FUNCTION_BLOCK "Driver_Working"   // FB15, SCL
{ S7_Optimized_Access := 'TRUE' }
VERSION : 0.1
   VAR_INPUT
      in_bStartButtonPushed : Bool;
      in_bEnableReturnTask : Bool;   // Включение. Режима добора задания
      in_bCountTriesReset : Bool;   // Сброс количества попыток перекладки
      in_usiCountTries : USInt;   // Количество попыток выполнить задание
      in_iRequired : Int;   // Задание. Кол-во материала
      in_bAlarm : Bool;   // Наличие Аварии
      in_bAlarmReset : Bool;   // Сброс Аварии
      in_bInHome : Bool;   // Сигнал от робота. Робот в Домашней позиции
      in_bProgReq : Bool;   // Сигнал от робота. Запрос на новую программу
      in_bResume : Bool;   // Продолжить выполнения задания
      in_bCancelTask : Bool;   // Отмена задания
      in_bModeDebug : Bool;   // Режим. Отладки
      in_pointer_array : Array[0..1] of Bool;
   END_VAR
   VAR_OUTPUT
      out_bStart : Bool;   // Команда Старт
      out_bStop : Bool;   // Команда Стоп
      out_usiProgrammNumber : USInt;   // Номер программы
      out_uiZoneFrom : UInt;   // Задание. Откуда забирать материал
      out_uiZoneTo : UInt;   // Задание. Куда класть материал
      out_uiRequired : UInt;   // Задание. Кол-во материала
      out_A_bCantWork : Bool;   // Авария Робот не может продолжать работу
      out_usiCountTries : USInt;   // Количество попыток
      out_strJobStatus : String[15];   // Статус задачи
   END_VAR
   VAR_IN_OUT
      in_Task : "TypeRobotTask";   // Собранное задание
      in_usiTaskStatus : UInt;   // Состояние Задания
      in_bDebugNextStep : Bool;   // Режим отладки. Следующий шаг
   END_VAR
   VAR
      _bStart : Bool;   // Бит старта Робота
      _bStop : Bool;   // Бит стоп Робота
      _uiZoneFrom : UInt;   // Задание. Откуда забирать материал
      _uiZoneTo : UInt;   // Задание. Куда класть материал
      _uiRequired : Int;   // Задание. Кол-во материала
      _bCancelTask : Bool;
      _usiStatus : USInt;
      _uiProgrammNumber : UInt;   // Номер программы
      _usiLastProgrammNumber : USInt;   // Последний номер программы
      _usiCountTries : USInt;   // Счетчик попыток
      _usiCountTriesHeight : USInt;
      _usiStepRegularWork : USInt;
      tStepBHX_scan : Array[0..17] of TON_TIME;
      i_tStepBHX_scan : USInt;
      tStepRegularWork : Array[0..17] of TON_TIME;
      i_tStepRegularWork : USInt;
      _usiStepCancelTask : USInt;
      tStepCancelTask : Array[0..17] of TON_TIME;
      i_tStepCancelTask : USInt;
      _usiStepAlaram : USInt;
      tStepAlaram : Array[0..17] of TON_TIME;
      i_tStepAlaram : USInt;
      rtFinish : R_TRIG;   // Тригер окончания задания
      rtAlarmReset : R_TRIG;   // Тригер продолжения задания
      rtCountTries : R_TRIG;   // Тригер счетчик попыток выполнения задания
      rtCountTriesReset : R_TRIG;   // Тригер сброса попыток выполнения задания
      rtStartButtonPushed : R_TRIG;
      _robot_status_ok : Bool;
      _part_status_ok : Bool;
      _task_status_ok : Bool;
      _robot_signals_ok : Bool;
      _first_step_ok : Bool;
      _act_done : Bool;
      _select_done : Bool;
      _task_id_ok : Bool;
      _lrobot_task_id : LInt;
   END_VAR
   VAR CONSTANT
      cTaskStatus_Ready : USInt := 0;   // Статус задания. Готов
      cTaskStatus_NewTaskReceived : USInt := 1;   // Статус задания. Получено новое задание
      cTaskStatus_InProcess : USInt := 2;   // Статус задания. В процессе
      cTaskStatus_Finished : USInt := 3;   // Статус задания. Закончено
      cWorkStatus_RegularWork : USInt := 99;   // Режим. Нормальная работа
      cWorkStatus_CancelTask : USInt := 1;   // Режим. Возврат в дом
      cWorkStatus_Alarm : USInt := 0;   // Режим. Авария
      cStep_ReadyForNewCyrcle : USInt := 0;   // Готовностьи к новому циклу
      cStep_SetRegularWorkProgramm : USInt := 1;   // Изменяем номер программы
      cStep_StartBitUp : USInt := 2;   // Выставляем стартовый бит
      cStep_StartBitDown : USInt := 3;   // Снимаем стартовый бит
      cStep_InProcess : USInt := 4;   // Переводим состояние задания в вПроцессе
      cStep_TaskFinish : USInt := 5;   // Задание завершенно
      cStep_DelayBeforeHome : USInt := 6;   // Ждем новое задание перед отправкой в дом
      cStep_SetGoHomeProgramm : USInt := 7;   // Отправляем робота в дом
      cStep_StartBitUpGoHome : USInt := 8;   // Выставляем стартовый бит
      cStep_StartBitDownGoHome : USInt := 9;   // Снимаем стартовый бит
      cStep_SendStopUp : USInt := 11;   // Выставляем Стоповый бит
      cStep_SendStopDown : USInt := 12;   // Снимаем Стоповый бит
      cStep_SetInitProgramm : USInt := 13;
      cStep_SetDeInitProgramm : USInt := 14;
      cStep_SetPostCorrProgramm : USInt := 15;
      cStep_StopBitUpGoHome : USInt := 16;
      cStep_StopBitDownGoHome : USInt := 17;
      cWorkStatus_Scanning : USInt := 2;   // Режим. Сканирование поддона
      cWorkStatus_HeightMeasuring : USInt := 3;
      cWorkStatus_Gripping_in : USInt := 4;
      cWorkStatus_Loading : USInt := 5;
      cWorkStatus_Unoading : USInt := 6;
      cWorkStatus_Flipping : USInt := 7;
      cWorkStatus_Dropping_out : USInt := 8;
      cWorkStatus_BHX_load : USInt := 9;
      cWorkStatus_BHX_unload : USInt := 10;
      cWorkStatus_BHX_scan : USInt := 11;
      cWorkStatus_test_BHX_load : USInt := 12;
      cWorkStatus_test_BHX_unload : USInt := 13;
      cWorkStatus_POS_load : USInt := 14;
      cWorkStatus_POS_unload : USInt := 15;
      cWorkStatus_Gripping_buf : USInt := 16;
      cWorkStatus_Dropping_buf : USInt := 17;
      cWorkStatus_Gripping_flip : USInt := 18;
      cWorkStatus_Dropping_flip : USInt := 19;
      cRange_k : Real := 0.0405;
      cRange_b : Real := 213.0;
   END_VAR
BEGIN
   ////////////////////////////Защиты и Блокировки////////////////////////////
   //Счетчик попыток на выполнение задания
   #rtCountTries(CLK := #_usiStepRegularWork = 1);
   IF #rtCountTries.Q THEN
       #_usiCountTries := #_usiCountTries + 1;
       #_usiCountTriesHeight := #_usiCountTriesHeight + 1;
   END_IF;
   #rtCountTriesReset(CLK := #in_bCountTriesReset);
   #rtAlarmReset(CLK := #in_bResume);
   IF #rtCountTriesReset.Q OR #rtAlarmReset.Q THEN
       #_usiCountTries := 0;
       #_usiCountTriesHeight := 0;
       #out_A_bCantWork := FALSE;
   END_IF;
   IF #_usiCountTries > (#in_usiCountTries) THEN
       #out_A_bCantWork := TRUE;
   END_IF;
   ///////////////////////////////////////////////////////////////////////////


   //
   #rtStartButtonPushed(CLK := #in_bStartButtonPushed AND (#_usiStepRegularWork < 1 OR #_usiStepRegularWork > 4));
   IF #rtStartButtonPushed.Q THEN
       #in_usiTaskStatus := 1;
   END_IF;

   //////////////////////////////Выбор состояния//////////////////////////////
   IF #in_bAlarm THEN
       //Статус: Авария 
       #_usiStatus := #cWorkStatus_Alarm;
   ELSIF (#in_bCancelTask OR #_bCancelTask) AND NOT #in_bAlarm THEN
       //Статус: Возврат в Дом 
       #_usiStatus := #cWorkStatus_CancelTask;
   ELSIF #in_bProgReq AND NOT #_bCancelTask AND NOT #in_bAlarm THEN //AND "PLC_AutoFeedingModeActive" THEN
       //Статус. Нормальный режим работы
       #_usiStatus := #cWorkStatus_RegularWork;
   ELSE
       #_uiProgrammNumber := 0;
   END_IF;
   ///////////////////////////////////////////////////////////////////////////

   ///////////////////////////////Логика работы///////////////////////////////
   //Статус: Нормальный режим работы
   IF #_usiStatus = #cWorkStatus_RegularWork THEN
       #rtFinish(CLK := #in_bProgReq);

       #_first_step_ok:=(#tStepRegularWork[#cStep_DelayBeforeHome].ET > T#20ms
                           OR #_usiStepRegularWork = #cStep_ReadyForNewCyrcle
                           OR (#_usiStepRegularWork = #cStep_SetRegularWorkProgramm AND #_uiProgrammNumber=0)
                           OR #tStepRegularWork[#cStep_StartBitDownGoHome].ET >= T#5s
                           OR "Robot"."EXT_FIRST_START")
                           AND #in_bProgReq
                           AND NOT "Robot"."PRO_MOVE_KRC";
                           #_task_status_ok := "RobotTasks".Robot1.task_status = 'received' OR "RobotTasks".Robot1.task_status = 'on_trajectory'
                           ;//OR "RobotTasks".Robot1.task_status = 'new_trajectory';
                           #_robot_status_ok := ("RobotTasks".Robot1.robot_status <> 'unknown') AND "RobotTasks".Robot1.robot_status <> 'manual_mode' AND "RobotTasks".Robot1.robot_status <> 'busy';
                           #_part_status_ok := ("RobotTasks".Robot1.part_status <> 'scanned'  OR "RobotTasks".Robot1.operation_type='measuring_height') AND "RobotTasks".Robot1.part_status <> 'done';

                           #_robot_signals_ok := "Robot"."USER_SAF_KRC" AND "Robot"."ALARM_STOP_KRC"  AND "Robot"."PERI_RDY_KRC" AND NOT "Robot"."STOPMESS_KRC" AND NOT "To_KUKA_PLC_STOP";

       #_task_id_ok:=#_lrobot_task_id="RobotTasks".Robot1.robot_task_id;

       //Шаг: Готовность
       IF #_first_step_ok AND #_task_status_ok AND #_robot_status_ok AND #_part_status_ok
           AND NOT #_select_done THEN
           #_lrobot_task_id := "RobotTasks".Robot1.robot_task_id;
           #_usiStepRegularWork := #cStep_ReadyForNewCyrcle;
       END_IF;

       //Шаг: Изменяем номер программы
       IF  // #rtFinish.Q AND
           #tStepRegularWork[#cStep_ReadyForNewCyrcle].ET > T#20ms AND
           #in_bProgReq THEN
           #_usiStepRegularWork := #cStep_SetRegularWorkProgramm;
       END_IF;

       //Шаг: Выставляем стартовый бит
       IF #tStepRegularWork[#cStep_SetRegularWorkProgramm].ET > T#20ms 
           AND #_uiProgrammNumber>0
           //machine shunt
           AND (NOT "RobotTasks".Robot1."w/o_machine_mode"
           OR ("RobotTasks".Robot1.robot_trajectory <> 'LoadMachine' OR "RobotTasks".Robot1.robot_trajectory <> 'UnloadMachine' )
           //OR (#_uiProgrammNumber<>7 AND #_uiProgrammNumber<>8)
           )
           //#_usiStepRegularWork = #cStep_SetRegularWorkProgramm AND
           AND #in_bProgReq THEN
           #_usiStepRegularWork := #cStep_StartBitUp;
       END_IF;

       //Шаг: Снимаем стартовый бит
       IF #tStepRegularWork[#cStep_StartBitUp].ET > T#20ms
           THEN

               #_usiStepRegularWork := #cStep_StartBitDownGoHome;
       END_IF;

       //Шаг: Переводим состояние задания в вПроцессе
       IF #tStepRegularWork[#cStep_StartBitDownGoHome].ET > T#20ms 
           AND NOT #in_bProgReq
           //AND "RobotTasks".Robot1.robot_status <> 'home'
       THEN
           #_usiStepRegularWork := #cStep_InProcess;
           #_act_done := FALSE;
       END_IF;

       //Шаг: Переводим состояние задания в в начало
       IF (#tStepRegularWork[#cStep_StartBitDownGoHome].ET >= T#1m
           //machine shunt
           OR (#tStepRegularWork[#cStep_InProcess].ET >= T#1ms AND "RobotTasks".Robot1."w/o_machine_mode"))
           AND #in_bProgReq AND "RobotTasks".Robot1.robot_alarm_reset
       THEN
           #_usiStepRegularWork := #cStep_ReadyForNewCyrcle;
       END_IF;

       //Шаг: Задание завершенно
       IF (#tStepRegularWork[#cStep_InProcess].ET > T#20ms
           //machine shunt
           OR ("RobotTasks".Robot1."w/o_machine_mode" AND ("RobotTasks".Robot1.robot_trajectory = 'LoadMachine' OR "RobotTasks".Robot1.robot_trajectory = 'UnloadMachine')
           //OR ("RobotTasks".Robot1."w/o_machine_mode" AND (#_uiProgrammNumber=7 OR #_uiProgrammNumber=8)
                   AND #tStepRegularWork[#cStep_SetRegularWorkProgramm].ET > T#20ms
               ))
               AND #in_bProgReq
               //AND ROR(IN := "Robot"."PGNO_REFL_KRC", N := 8) = #_uiProgrammNumber
       THEN
           #_usiStepRegularWork := #cStep_TaskFinish;
           #_act_done := FALSE;
       END_IF;

       //Шаг: Переход к ожиданию нового цикла
       IF  #tStepRegularWork[#cStep_TaskFinish].ET > T#500ms OR "To_KUKA_PLC_STOP" THEN
           #_usiStepRegularWork := #cStep_DelayBeforeHome;
           #_uiProgrammNumber := 0;
       END_IF;

       CASE #_usiStepRegularWork OF
           #cStep_ReadyForNewCyrcle:
               //Шаг: Готовность
               #_bStart := FALSE;
               #_uiProgrammNumber := 0;

           #cStep_SetRegularWorkProgramm:
               //Шаг: Изменяем номер программы
               IF #_uiProgrammNumber = 0 THEN
                   "Get_Robot_Program"(in_Task:="RobotTasks".Robot1, Program_number=>#_uiProgrammNumber );
                   IF #_uiProgrammNumber <> 0 THEN
                       IF "RobotTasks".Robot1.part_status = 'ordered' THEN
                           "To_KUKA_Part_Destination" := 1;
                       ELSIF "RobotTasks".Robot1.part_status = 'processing' THEN
                           "To_KUKA_Part_Destination" := 2;
                       ELSIF "RobotTasks".Robot1.part_status = 'loading' THEN
                           "To_KUKA_Part_Destination" := 3;
                       ELSIF "RobotTasks".Robot1.part_status = 'unloading' THEN
                           "To_KUKA_Part_Destination" := 4;
                       ELSIF "RobotTasks".Robot1.part_status = 'done' THEN
                           "To_KUKA_Part_Destination" := 5;
                       ELSIF "RobotTasks".Robot1.part_status = 'in_machine' THEN
                           "To_KUKA_Part_Destination" := 6;
                       ELSIF "RobotTasks".Robot1.part_status = 'pallet_in' THEN
                           "To_KUKA_Part_Destination" := 7;
                       ELSIF "RobotTasks".Robot1.part_status = 'pallet_buf' THEN
                           "To_KUKA_Part_Destination" := 8;
                       ELSIF "RobotTasks".Robot1.part_status = 'pallet_out' THEN
                           "To_KUKA_Part_Destination" := 9;
                       ELSIF "RobotTasks".Robot1.part_status = 'gripper' THEN
                           "To_KUKA_Part_Destination" := 10;
                       ELSIF "RobotTasks".Robot1.part_status = 'grabbing' THEN
                           "To_KUKA_Part_Destination" := 11;
                       ELSIF "RobotTasks".Robot1.part_status = 'dropping' THEN
                           "To_KUKA_Part_Destination" := 12;
                       ELSIF "RobotTasks".Robot1.part_status = 'scanning' THEN
                           "To_KUKA_Part_Destination" := 13;
                       ELSIF "RobotTasks".Robot1.part_status = 'part_slot' THEN
                           "To_KUKA_Part_Destination" := 14;
                       ELSIF "RobotTasks".Robot1.part_status = 'flip_table' THEN
                           "To_KUKA_Part_Destination" := 15;
                       ELSIF "RobotTasks".Robot1.part_status = 'flipping' THEN
                           "To_KUKA_Part_Destination" := 16;
                       ELSIF "RobotTasks".Robot1.part_status = 'scanned' THEN
                           "To_KUKA_Part_Destination" := 17;
                       ELSIF "RobotTasks".Robot1.part_status = 'measuring' THEN
                           "To_KUKA_Part_Destination" := 18;
                       END_IF;
                       "RobotTasks".Robot1.robot_program:=#_uiProgrammNumber;
                       "RobotTasks".Robot1.robot_trajectory:="Robot_Programs".List[#_uiProgrammNumber].trajectory;
                       //"RobotTasks".Robot1.task_status:='new_trajectory';
                   END_IF;
               END_IF;

           #cStep_StartBitUp:
               //Шаг: Выставляем стартовый бит
               #_bStart := TRUE;

           #cStep_StartBitDownGoHome:
               //Шаг: Снимаем стартовый бит
               #_bStart := FALSE;

           #cStep_InProcess:
               //Шаг: Переводим состояние задания в вПроцессе
               IF "RobotTasks".Robot1.robot_trajectory = 'PartHeightMeasuring' AND
                   #tStepRegularWork[#cStep_InProcess].ET > T#200ms AND NOT "Robot"."PRO_MOVE_KRC" THEN
                   "RobotTasks".Robot1.part_pos_Z := "Robot".POS_ACT_Z - ("InGripperRangefinder" * #cRange_k + #cRange_b);
                   "RobotTasks".Robot1.slot_pos_Z := ("InGripperRangefinder" * #cRange_k + #cRange_b);
               END_IF;
               IF "Robot_Programs".List["RobotTasks".Robot1.robot_program].OUT_Status.inprocess_part_status = '' THEN
                   CASE "Robot"."Part_Status" OF
                       1:  "RobotTasks".Robot1.part_status := 'ordered';
                       2:  "RobotTasks".Robot1.part_status := 'processing';
                       3:  "RobotTasks".Robot1.part_status := 'loading';
                       4:  "RobotTasks".Robot1.part_status := 'unloading';
                       5:  "RobotTasks".Robot1.part_status := 'done';
                       6:  "RobotTasks".Robot1.part_status := 'in_machine';
                       7:  "RobotTasks".Robot1.part_status := 'pallet_in';
                       8:  "RobotTasks".Robot1.part_status := 'pallet_buf';
                       9:  "RobotTasks".Robot1.part_status := 'pallet_out';
                       10: "RobotTasks".Robot1.part_status := 'gripper';
                       11: "RobotTasks".Robot1.part_status := 'grabbing';
                       12: "RobotTasks".Robot1.part_status := 'dropping';
                       13: "RobotTasks".Robot1.part_status := 'scanning';
                       14: "RobotTasks".Robot1.part_status := 'part_slot';
                       15: "RobotTasks".Robot1.part_status := 'flip_table';
                       16: "RobotTasks".Robot1.part_status := 'flipping';
                       17: "RobotTasks".Robot1.part_status := 'scanned';
                       18: "RobotTasks".Robot1.part_status := 'measuring';
                   END_CASE;
               END_IF;

               IF NOT #_act_done AND #_robot_signals_ok AND #_task_id_ok THEN
                   //IF "RobotTasks".Robot1.robot_trajectory = 'PutOnSlot' THEN
                   //"RobotTasks".Robot1.part_slot := "RobotTasks".Robot1.free_slot;
                   //END_IF;
                   "RobotTasks".Robot1.task_status := "Robot_Programs".List["RobotTasks".Robot1.robot_program].OUT_Status.inprocess_task_status;
                   IF "Robot_Programs".List["RobotTasks".Robot1.robot_program].OUT_Status.inprocess_part_status <> '' THEN
                       "RobotTasks".Robot1.part_status := "Robot_Programs".List["RobotTasks".Robot1.robot_program].OUT_Status.inprocess_part_status;
                   END_IF;
                   #_act_done := TRUE;
               END_IF;

           #cStep_TaskFinish:
               //Шаг: Задание завершенно
               IF NOT #_act_done AND #_robot_signals_ok AND #_task_id_ok THEN
                   IF "RobotTasks".Robot1.robot_trajectory = 'PutOnFlipTableB' OR "RobotTasks".Robot1.robot_trajectory = 'AutoMachiningA_' THEN
                       IF "RobotTasks".Robot1.part_side = 'A' THEN
                           "RobotTasks".Robot1.part_side := 'B';
                       ELSIF "RobotTasks".Robot1.part_side = 'B' THEN
                           "RobotTasks".Robot1.part_side := 'A';
                       END_IF;
                   END_IF;
                   IF "RobotTasks".Robot1.robot_trajectory = 'PartHeightMeasuring' THEN
                       "RobotTasks".Robot1.part_pos_Z := "Robot".POS_ACT_Z - ("InGripperRangefinder" * #cRange_k + #cRange_b);
                       "RobotTasks".Robot1.slot_pos_Z := ("InGripperRangefinder" * #cRange_k + #cRange_b);
                   END_IF;
                   IF "RobotTasks".Robot1.robot_trajectory = 'Pallet_Scanning' THEN
                       "Matrix_output".scan_lay_number := "Matrix_output".scan_lay_number + 1;
                   END_IF;
                   IF "RobotTasks".Robot1.robot_trajectory = 'TakeFromSlot' THEN
                       "RobotTasks".Robot1.part_slot := 0;
                   END_IF;
                   //Не тот слой
                   IF "RobotTasks".Robot1.robot_trajectory = 'TakeFromPalletIn' AND NOT "Robot"."PartOK" THEN
                       //"RobotTasks".Robot1.task_status := 'not_sended';
                       //"RobotTasks".Robot1.part_status := 'ordered';
                       ;
                   END_IF;
                   "RobotTasks".Robot1.task_status := "Robot_Programs".List["RobotTasks".Robot1.robot_program ].OUT_Status.finish_task_status;
                   IF "Robot_Programs".List["RobotTasks".Robot1.robot_program].OUT_Status.finish_part_status <> '' THEN
                       "RobotTasks".Robot1.part_status := "Robot_Programs".List["RobotTasks".Robot1.robot_program].OUT_Status.finish_part_status;
                    END_IF;
                   #_act_done := TRUE;
               END_IF;
       END_CASE;
   END_IF;

   //Статус: Отмена задания и возврат в дом
   IF #_usiStatus = #cWorkStatus_CancelTask THEN
       //Шаг: Отправляем на робота команду стоп (для выхода из программы)
       IF #_usiStepCancelTask = #cStep_ReadyForNewCyrcle OR #in_bCancelTask THEN
           #_usiStepCancelTask := #cStep_SendStopUp;
       END_IF;

       //Шаг: Снимаем команду стоп
       IF #tStepCancelTask[#cStep_SendStopUp].ET > T#300ms THEN
           #_usiStepCancelTask := #cStep_SendStopDown;
       END_IF;

       //Шаг: Изменяем номер программы
       IF #tStepCancelTask[#cStep_SendStopDown].ET > T#200ms THEN
           #_usiStepCancelTask := #cStep_SetGoHomeProgramm;
       END_IF;

       //Шаг: Отправляем стартовый бит
       IF #tStepCancelTask[#cStep_SetGoHomeProgramm].ET > T#300ms THEN
           #_usiStepCancelTask := #cStep_StartBitUpGoHome;
       END_IF;

       //Шаг: Снимаем стартовый бит
       IF #tStepCancelTask[#cStep_StartBitUpGoHome].ET > T#300ms OR #in_bInHome THEN
           #_usiStepCancelTask := #cStep_StartBitDownGoHome;
       END_IF;

       CASE #_usiStepCancelTask OF
           #cStep_SendStopUp:
               //Шаг: Отправляем на робота команду стоп(для выхода из программы в CELL) и сбрасываем вакуум
               #_bStop := TRUE;
               #_bCancelTask := TRUE;

           #cStep_SendStopDown:
               //Шаг: Снимаем команду стоп и срос вакуума
               #_bStop := FALSE;

           #cStep_SetGoHomeProgramm:
               //Шаг: Изменяем номер программы
               #_uiProgrammNumber := 10;

           #cStep_StartBitUpGoHome:
               //Шаг: Отправляем стартовый бит
               #_bStart := TRUE;

           #cStep_StartBitDownGoHome:
               //Шаг: Снимаем стартовый бит
               #_bStart := FALSE;
               #_bCancelTask := FALSE;
       END_CASE;
   ELSE
       #_usiStepCancelTask := 0;
       #_bCancelTask := FALSE;
       #_bStop := FALSE;
   END_IF;

   //Статус: Авария, Возврат в дом
   IF #_usiStatus = #cWorkStatus_Alarm THEN
       //Шаг: Изменяем номер программы
       IF  #_usiStepAlaram = 0 AND #in_bAlarmReset THEN
           #_usiStepAlaram := #cStep_SetGoHomeProgramm;
       END_IF;

       //Шаг: Отправляем стартовый бит
       IF #tStepAlaram[#cStep_SetGoHomeProgramm].ET > T#20ms THEN
           #_usiStepAlaram := #cStep_StartBitUpGoHome;
       END_IF;

       //Шаг: Снимаем стартовый бит
       IF #tStepAlaram[#cStep_StartBitUpGoHome].ET > T#20msTHEN
           #_usiStepAlaram := #cStep_StartBitDownGoHome;
       END_IF;

       CASE #_usiStepAlaram OF
           #cStep_SetGoHomeProgramm:
               //Шаг: Изменяем номер программы
               #_uiProgrammNumber := 100;

           #cStep_StartBitUpGoHome:
               //Шаг: Отправляем стартовый бит
               #_bStart := TRUE;

           #cStep_StartBitDownGoHome:
               //Шаг: Снимаем стартовый бит
               #_bStart := FALSE;
       END_CASE;
   ELSE
       #_usiStepAlaram := 0;
   END_IF;

   ///////////////////////////////////////////////////////////////////////////

   ///////////////////////////////Запись выходов//////////////////////////////
   IF #_uiProgrammNumber<>0 THEN
       #_usiLastProgrammNumber := #_uiProgrammNumber;
   END_IF;
   #out_usiProgrammNumber := #_uiProgrammNumber;
   #out_bStart := #_bStart;
   #out_bStop := #_bStop;
   #out_uiZoneFrom := #_uiZoneFrom;
   #out_uiZoneTo := #_uiZoneTo;
   #out_uiRequired := #_uiRequired;
   #out_usiCountTries := #_usiCountTries;
   ///////////////////////////////////////////////////////////////////////////

   //////////////////////////////////Таймеры//////////////////////////////////
   //Запуск
   #tStepRegularWork[#_usiStepRegularWork](IN := TRUE,
                                           PT := T#1m);
   #tStepCancelTask[#_usiStepCancelTask](IN := TRUE,
                                             PT := T#1m);
   #tStepAlaram[#_usiStepAlaram](IN := TRUE,
                                 PT := T#1m);
   //Сброс
   FOR #i_tStepRegularWork := 0 TO 17 DO
       IF #_usiStepRegularWork <> #i_tStepRegularWork THEN
           #tStepRegularWork[#i_tStepRegularWork](IN := FALSE,
                                                  PT := T#10s);
       END_IF;
   END_FOR;
   FOR #i_tStepCancelTask := 0 TO 15 DO
       IF #_usiStepCancelTask <> #i_tStepCancelTask THEN
           #tStepCancelTask[#i_tStepCancelTask](IN := FALSE,
                                                PT := T#10s);
       END_IF;
   END_FOR;
   FOR #i_tStepAlaram := 0 TO 15 DO
       IF #_usiStepAlaram <> #i_tStepAlaram THEN
           #tStepAlaram[#i_tStepAlaram](IN := FALSE,
                                        PT := T#10s);
       END_IF;
   END_FOR;
   ///////////////////////////////////////////////////////////////////////////
END_FUNCTION_BLOCK

// folder: 5_Matrix_scanner

FUNCTION_BLOCK "DADProtocol"   // FB2, SCL
{ S7_Optimized_Access := 'TRUE' }
VERSION : 0.1
   VAR_INPUT
      DAD_ENABLE : Bool;
      IOconditioning_Enable : Bool;   // User should edit this parameter according to the Reader configuration in DL.CODE
      DataConsistency_Enable : Bool;   // User should edit this parameter according to the Reader configuration in DL.CODE
      OutputExArea_FirstByteAddress : Int;   // User should edit this parameter according to the Reader Output Exchange area addresses
      OutputExArea_Size : Int;   // User should edit this parameter according to the Reader Output Exchange area size
      InputExArea_FirstByteAddress : Int;   // User should edit this parameter according to the Reader Input Exchange area addresses
      InputExArea_Size : Int;   // User should edit this parameter according to the Reader Input Exchange area size
   END_VAR
   VAR_OUTPUT
      newDataBlockReceived : Bool;
      newDataBlockLength : Int;
   END_VAR
   VAR_IN_OUT
      Do_Resync : Bool;
      Do_SendData : Bool;
      DataToSendLength : Byte;
   END_VAR
   VAR
      newInputDataAvailable : Bool;
      InputExArea_Type : Byte := 16#81;   // User should edit this parameter according to the Reader Input Exchange area type. 16#81 --> Input ; 16#82 --> Output ; 16#84 --> DB
      OutputExArea_Type : Byte := 16#82;   // User should edit this parameter according to the Reader Output Exchange area type. 16#81 --> Input ; 16#82 --> Output ; 16#84 --> DB
      DB_Number : DInt;   // If the Exchange Area type is 16#84 (DB), this parameter specifies the DB number
      inputBuffer : Array[0..512] of Byte;
      outputBuffer : Array[0..512] of Byte;
      DAD_PRTL_FIRST_ITERATION : Bool := true;
      DAD_InternalStates : Int;
      AddressOffset : Int;
      InputDataLenByteAddress : Int;
      InputControlByteAddress : Int;
      InputFirstDataByteAddress : Int;
      InputDataConistencyByteAddress : Int;
      InputDataByteAddress : Int;
      InputDataAvailable_Actual : Bool;
      InputFragmentedData_Actual : Bool;
      InputFragmentedData_Previous : Bool;
      InputDeviceDadEnable : Bool;
      InputResyncAck : Bool;
      InputControlByte : Byte;
      InputDataLength : Byte;
      InputDataConsistencyByte : Byte;
      DataByteIndex : Int;
      OutputControlByteAddress : Int;
      OutputControlByte : Byte;
      OutputDataConsistencyByteAddress : Int;
      OutputAckDataReceived : Bool;
      TempByteValue : Byte;
      BufferDataByteIndex : Int;
      BeginFragmentedDataRx : Bool;
      EndFragmentedDataRx : Bool;
      FragmentedDataRxEnable : Bool;
      DataFragmentIndex : Int;
      MaxInputFragmentDimension : Int;
      DAD_PRTL_NUM_BYTE : Int;
      IO_COND_NUM_BYTE : Int;
      DATA_CONSISTENCY_NUM_BYTE : Int;
      Error_INPUT_DATA_CONSISTENCY : Bool;
      Error_DAD_DISABLED_ON_DEVICE : Bool;
      OutputDataLenByteAddress : Int;
      OutputFirstDataByteAddress : Int;
      NewMessageReady : Bool;
      ackDataReceived : Bool;
   END_VAR
   VAR_TEMP
      MessageByteIndex : Int;
      resetByte : Byte;
   END_VAR
   VAR CONSTANT
      IDLE : Int := 0;
      WAIT_DEVICE_DAD_ENABLING : Int := 1;
      CHECK_DATA_CONSISTENCY : Int := 10;
      READ_DATA : Int := 20;
      SEND_DATA : Int := 40;
      WAIT_ACK_DATA_SENT : Int := 41;
      SEND_SYNC_REQUEST : Int := 30;
      WAIT_SYNC_ACK : Int := 31;
      SEND_END_SYNC_REQUEST : Int := 32;
      WAIT_END_SYNC_ACK : Int := 33;
   END_VAR
BEGIN
   IF #DAD_ENABLE THEN
       // IF THE DAD PROTOCOL IS ENABLED..

       IF #DAD_PRTL_FIRST_ITERATION THEN

           // ONLY DURING THE FIRST ITERATION AFTER DAD PROTOCOL ENABLING...

           (*------------------------------------------------------------------------------
           ********************* PROTOCOL INITIALIZATION PHASE ****************************
           --------------------------------------------------------------------------------

           The Protocol initializes its parameters AND sets the Bit 7 of the Output Control
           Byte.

           ================================================================================
           Depending on the configuration parameters the addresses of the Protocol Bytes 
           varies. Suppose an Exchange Area of N Bytes. If DAD, I/O condtioning, and Data
           Consistency are enabled then the position of the bytes inside the data frame 
           will be the following.

               BYTEs POSITIONs     BYTEs Desriptions  

           |         0         | I/0 Conditioning      |
           |         1         | DAD CTRL Byte         |
           |         2         | DAD SAP Byte          |
           |         3         | DAD LENGTH Byte       |
           |      4 -> N-2     | DATA                  |
           |        N-1        | DATA CONSISTENCY Byte |

           ================================================================================*)

           #DAD_PRTL_NUM_BYTE              := 3;

           IF #IOconditioning_Enable THEN
               // If I/O conditioning is actiated the I/O data is shifted forward by one byte
               #IO_COND_NUM_BYTE           := 1;
           END_IF;

           IF #DataConsistency_Enable THEN
               // If I/O conditioning is actiated the last Byte of the Exchange area will
               // contain the copy of the DAD Control Byte
               #DATA_CONSISTENCY_NUM_BYTE          := 1;
               #InputDataConistencyByteAddress     := #InputExArea_FirstByteAddress + #InputExArea_Size - 1;
               #OutputDataConsistencyByteAddress   := #OutputExArea_FirstByteAddress + #OutputExArea_Size - 1;
           END_IF;

           // Effective dimension of the data which can be received
           #MaxInputFragmentDimension      := #InputExArea_Size - #IO_COND_NUM_BYTE - #DATA_CONSISTENCY_NUM_BYTE - #DAD_PRTL_NUM_BYTE;

           #InputControlByteAddress        := #InputExArea_FirstByteAddress + #IO_COND_NUM_BYTE;
           #InputDataLenByteAddress        := #InputExArea_FirstByteAddress + #IO_COND_NUM_BYTE + 2;
           #InputFirstDataByteAddress      := #InputExArea_FirstByteAddress + #IO_COND_NUM_BYTE + 3;
           #OutputControlByteAddress       := #OutputExArea_FirstByteAddress + #IO_COND_NUM_BYTE;
           #OutputDataLenByteAddress       := #OutputExArea_FirstByteAddress + #IO_COND_NUM_BYTE + 2;
           #OutputFirstDataByteAddress     := #OutputExArea_FirstByteAddress + #IO_COND_NUM_BYTE + 3;

           // DAD Output Bit Enable set to '1' by the protocol
           POKE_BOOL(area                  := #OutputExArea_Type,
                     byteOffset            := #OutputControlByteAddress,
                     bitOffset             := 7,
                     dbNumber              := #DB_Number,
                     value                 := TRUE);

           #newDataBlockReceived           := FALSE;
           #newDataBlockLength             := 0;

           #DAD_PRTL_FIRST_ITERATION       := FALSE;

           // !!! After enabling the DAD, the PLC performs a resynchronization with the device !!!
           #DAD_InternalStates             := #SEND_SYNC_REQUEST;

       ELSE

           // IF IT'S NOT THE FIRST ITERATION AFTER DAD PROTOCOL ENABLING....

           (* =================================================================================
           ------------------------------------------------------------------------------------

           1st Operation.                INPUT/OUTPUT SAMPLING 

           ----------------------------------------------------------------------------------
           ==================================================================================*)

           // Storing the Actual Values of the INPUT CONTROL BYTE's BITS OF INTEREST  

           #InputControlByte               := PEEK_BYTE(area := #InputExArea_Type, byteOffset := #InputControlByteAddress, dbNumber := #DB_Number);
           #InputDataAvailable_Actual      := #InputControlByte.%X0;
           #InputResyncAck                 := #InputControlByte.%X2;
           #InputFragmentedData_Actual     := #InputControlByte.%X3;
           #InputDeviceDadEnable           := #InputControlByte.%X7;
           #InputDataConsistencyByte       := PEEK_BYTE(area := #InputExArea_Type, byteOffset := #InputDataConistencyByteAddress, dbNumber := #DB_Number);

           // Storing the Actual Values of the OUTPUT CONTROL BYTE's BITS OF INTEREST
           #OutputControlByte              := PEEK_BYTE(area := #OutputExArea_Type, byteOffset := #OutputControlByteAddress, dbNumber := #DB_Number);
           #OutputAckDataReceived          := #OutputControlByte.%X0;
           //my huck
           //#InputResyncAck := FALSE;
           (*==================================================================================
           ++++++++++++++++++++++++++++++++++++++++++++++++++++++++++++++++++++++++++++++++++++

           2nd Operation.           BEGIN DAD FINITE STATES MACHINE

           ++++++++++++++++++++++++++++++++++++++++++++++++++++++++++++++++++++++++++++++++++++
           ==================================================================================*)

           CASE #DAD_InternalStates OF

                   (* ------------------------------------------------------------------------------------------
                   ********************************** PROTOCOL IDLE STATE **************************************
                   ---------------------------------------------------------------------------------------------

                   In the IDLE state the Protocol controls the input of the function block and the input control
                   Byte to determin which procedure has to be done *)

               0: // IDLE

                   // ========================= CHECK FOR NEW INPUT DATA =============================

                   #newInputDataAvailable              := #InputDataAvailable_Actual <> #OutputAckDataReceived;

                   IF #newInputDataAvailable THEN
                       // If a new Stream Of Data is available from the reader..
                       // Rising Edge of the Bit 3 in the Input CTRL Byte means Start Of FRAGMENTED Data Trasmission
                       #BeginFragmentedDataRx          := #InputFragmentedData_Actual AND NOT #InputFragmentedData_Previous;
                       // Falling Edge of the Bit 3 in the Input CTRL Byte means End Of FRAGMENTED Data Trasmission
                       #EndFragmentedDataRx            := NOT #InputFragmentedData_Actual AND #InputFragmentedData_Previous;

                       IF #BeginFragmentedDataRx THEN
                           // If the Data is Fragmented the Protocol prepares for receiving each fragment
                           #FragmentedDataRxEnable     := TRUE;
                           #DataFragmentIndex          := 0;
                       END_IF;

                       IF #DataConsistency_Enable THEN

                           // Protocol Verifies the consistency and THEN read the data
                           IF #InputControlByte = #InputDataConsistencyByte THEN
                               #Error_INPUT_DATA_CONSISTENCY       := FALSE;
                               #DAD_InternalStates                 := #READ_DATA;
                           ELSE
                               #Error_INPUT_DATA_CONSISTENCY       := TRUE;
                               // #DAD_InternalStates                 := #CHECK_DATA_CONSISTENCY;
                           END_IF;

                       ELSE

                           // Protocol Reads the data
                           #DAD_InternalStates                     := #READ_DATA;

                       END_IF;

                   END_IF;

                   #InputFragmentedData_Previous := #InputFragmentedData_Actual;


                   (*========================= USER ASKED FOR SENDING DATA ==========================
                      The Send Data procedure has higher priority than the reading data one
                   *)

                   IF #Do_SendData THEN
                       #DAD_InternalStates := #SEND_DATA;
                   END_IF;



                   (*=========================== USER ASKED FOR RESYNC ==============================
                      The Resynchronization procedure has higher priority than sending/reading data
                   *)

                   IF #Do_Resync THEN
                       #DAD_InternalStates                 := #SEND_SYNC_REQUEST;
                   END_IF;

                   (*=========================== DAD ON DEVICE IS OFF ===============================
                   If the device is down the protocol waits for its recover (DAD Bit sets to 1) and
                   automatically resync with it
                   *)

                   IF NOT #InputDeviceDadEnable THEN
                       #Error_DAD_DISABLED_ON_DEVICE       := TRUE;
                       #DAD_InternalStates                 := #WAIT_DEVICE_DAD_ENABLING;
                   END_IF;


                   (* --------------------------------------------------------------------------------------
                   ************************* PROTOCOL WAITS FOR DEVICE RECOVER *****************************
                   ----------------------------------------------------------------------------------------*)

               1: // WAIT_DEVICE_DAD_ENABLING

                   IF #InputDeviceDadEnable THEN
                       #Error_DAD_DISABLED_ON_DEVICE       := FALSE;
                       #DAD_InternalStates                 := #SEND_SYNC_REQUEST;
                   END_IF;


                   (* --------------------------------------------------------------------------------------
                   ******************************* PROTOCOL RECEIVES DATA ***********************************
                   ----------------------------------------------------------------------------------------*)

               20: // READ_DATA

                   #InputDataLength := PEEK_BYTE(area := #InputExArea_Type, byteOffset := #InputDataLenByteAddress, dbNumber := #DB_Number);

                   FOR #DataByteIndex := 0 TO BYTE_TO_INT(#InputDataLength) - 1 DO
                       #InputDataByteAddress           := #InputFirstDataByteAddress + #DataByteIndex;
                       #TempByteValue                  := PEEK_BYTE(area := #InputExArea_Type, byteOffset := #InputDataByteAddress, dbNumber := #DB_Number);
                       #BufferDataByteIndex            := #DataByteIndex + (#MaxInputFragmentDimension * #DataFragmentIndex);
                       #inputBuffer[#BufferDataByteIndex] := #TempByteValue;
                   END_FOR;

                   IF #FragmentedDataRxEnable THEN
                       // If the Fragmentation is Enabled i prepare for reading the next fragment
                       #DataFragmentIndex := #DataFragmentIndex + 1;

                       IF #EndFragmentedDataRx THEN
                           // If it has been received the last fragment the Protocol:
                           #newDataBlockReceived   := NOT #newDataBlockReceived;
                           #newDataBlockLength     := #BufferDataByteIndex + 1;
                           #FragmentedDataRxEnable := FALSE;       // Disable the Data Fragmentation Enable
                           #DataFragmentIndex      := 0;           // Reset the Data Fragment Index
                       END_IF;

                   ELSE
                       #newDataBlockReceived       := NOT #newDataBlockReceived;
                       #newDataBlockLength         := #BufferDataByteIndex + 1;
                   END_IF;

                   // SEND_ACKNOWLEDGE_DATA_READ

                   POKE_BOOL(area          := #OutputExArea_Type,
                             byteOffset    := #OutputControlByteAddress,
                             bitOffset     := 0,
                             dbNumber      := #DB_Number,
                             value         := #InputDataAvailable_Actual); // DAD Protocol send the Ack

                   #DAD_InternalStates     := #IDLE;

                   (* --------------------------------------------------------------------------------------
                   ************************* PROTOCOL RESYNCHRONIZES WITH DEVICE ***************************
                   ---------------------------------------------------------------------------------------*)

               30: // SEND_SYNC_REQUEST

                   POKE_BOOL(area          := #OutputExArea_Type,
                             byteOffset    := #OutputControlByteAddress,
                             bitOffset     := 2,
                             dbNumber      := #DB_Number,
                             value         := TRUE); // Protocol SET the Sync REQUEST

                   #DAD_InternalStates     := #WAIT_SYNC_ACK;

               31: // WAIT_SYNC_ACK

                   //Protocol Waits the Acknowledge from the Reader
                   IF #InputResyncAck THEN

                       POKE_BOOL(area          := #OutputExArea_Type,
                                 byteOffset    := #OutputControlByteAddress,
                                 bitOffset     := 1,
                                 dbNumber      := #DB_Number,
                                 value         := FALSE); // Protocol RESET the Output Data Ready Bit

                       POKE_BOOL(area          := #OutputExArea_Type,
                                 byteOffset    := #OutputControlByteAddress,
                                 bitOffset     := 0,
                                 dbNumber      := #DB_Number,
                                 value         := FALSE); // Protocol RESET the Input Data Received Bit

                       #DAD_InternalStates     := #SEND_END_SYNC_REQUEST;

                   END_IF;

               32: // SEND_END_SYNC_REQUEST

                   POKE_BOOL(area              := #OutputExArea_Type,
                             byteOffset        := #OutputControlByteAddress,
                             bitOffset         := 2,
                             dbNumber          := #DB_Number,
                             value             := FALSE); // Protocol RESET the Sync REQUEST

                   #DAD_InternalStates := #WAIT_END_SYNC_ACK;

               33: // WAIT_END_SYNC_ACK

                   IF NOT #InputResyncAck THEN
                       #Do_Resync       := FALSE;           // Reset the Resync command, so that operation is executed just one time
                       #DAD_InternalStates     := #IDLE;
                   END_IF;


                   (* --------------------------------------------------------------------------------------
                   ******************************** PROTOCOL SENDS DATA ************************************
                   ----------------------------------------------------------------------------------------*)

               40: // SEND_DATA

                   POKE(area := #OutputExArea_Type,
                        byteOffset := #OutputDataLenByteAddress,
                        dbNumber := 0,
                        value := #DataToSendLength);

                   FOR #MessageByteIndex := 0 TO BYTE_TO_INT(#DataToSendLength)-1 DO
                       POKE(area := #OutputExArea_Type,
                            byteOffset := #OutputFirstDataByteAddress + #MessageByteIndex,
                            dbNumber := 0,
                            value := #outputBuffer[#MessageByteIndex]);
                   END_FOR;

                   #NewMessageReady := NOT #NewMessageReady;

                   POKE_BOOL(area := #OutputExArea_Type,
                             byteOffset := #OutputControlByteAddress,
                             bitOffset := 1,
                             dbNumber := 0,
                             value := #NewMessageReady);

                   #DAD_InternalStates := 41;

               41: // WAIT_ACK_DATA_SENT

                   #ackDataReceived := PEEK_BOOL(area := #InputExArea_Type, dbNumber := 0, byteOffset := #InputControlByteAddress, bitOffset := 1);

                   IF #ackDataReceived = #NewMessageReady THEN
                       #Do_SendData := FALSE;
                       #DAD_InternalStates := #IDLE;
                   END_IF;



           END_CASE;// END STATES MACHINE

           (*==================================================================================
           ++++++++++++++++++++++++++++++++++++++++++++++++++++++++++++++++++++++++++++++++++++

                                      END DAD FINITE STATES MACHINE

           ++++++++++++++++++++++++++++++++++++++++++++++++++++++++++++++++++++++++++++++++++++
           ==================================================================================*)

       END_IF;// END FIRST ITERATION IF

       IF #DataConsistency_Enable THEN
           // IF DATA CONSISTENCY IS ENBLED:
           // The DAD Protocol copies the DAD CTRL Byte to the last byte position in the Out Exchange area.
           #OutputControlByte      := PEEK_BYTE(area := #OutputExArea_Type, byteOffset := #OutputControlByteAddress, dbNumber := #DB_Number);
           POKE(area               := #OutputExArea_Type,
                byteOffset         := #OutputDataConsistencyByteAddress,
                dbNumber           := #DB_Number,
                value              := #OutputControlByte);
       END_IF;

   ELSIF NOT #DAD_ENABLE & NOT #DAD_PRTL_FIRST_ITERATION THEN // IF THE DAD PROTOCOL IS DISABLED

       #resetByte              := 2#0000_0000;
       POKE(   area            := #OutputExArea_Type,
               byteOffset      := #OutputControlByteAddress,
               dbNumber        := #DB_Number,
               value           := #resetByte);

       #Do_Resync := FALSE;
       #Do_SendData := FALSE;
       #newDataBlockReceived := FALSE;
       #newDataBlockLength := 0;

       #DAD_PRTL_FIRST_ITERATION := TRUE;

   END_IF;// END DAD ENABLE IF
END_FUNCTION_BLOCK

FUNCTION "Matrix" : Void   // FC2, LAD
{ S7_Optimized_Access := 'TRUE' }
VERSION : 0.1
   VAR_TEMP
      RetVal : Word;
      PhaseON : DWord;
      PhaseOFF : DWord;
   END_VAR
   VAR_TEMP   // added for the SCL form of the ladder/FBD networks
      _w1 : Bool;
      _w2 : Bool;
   END_VAR
BEGIN

REGION Network 1
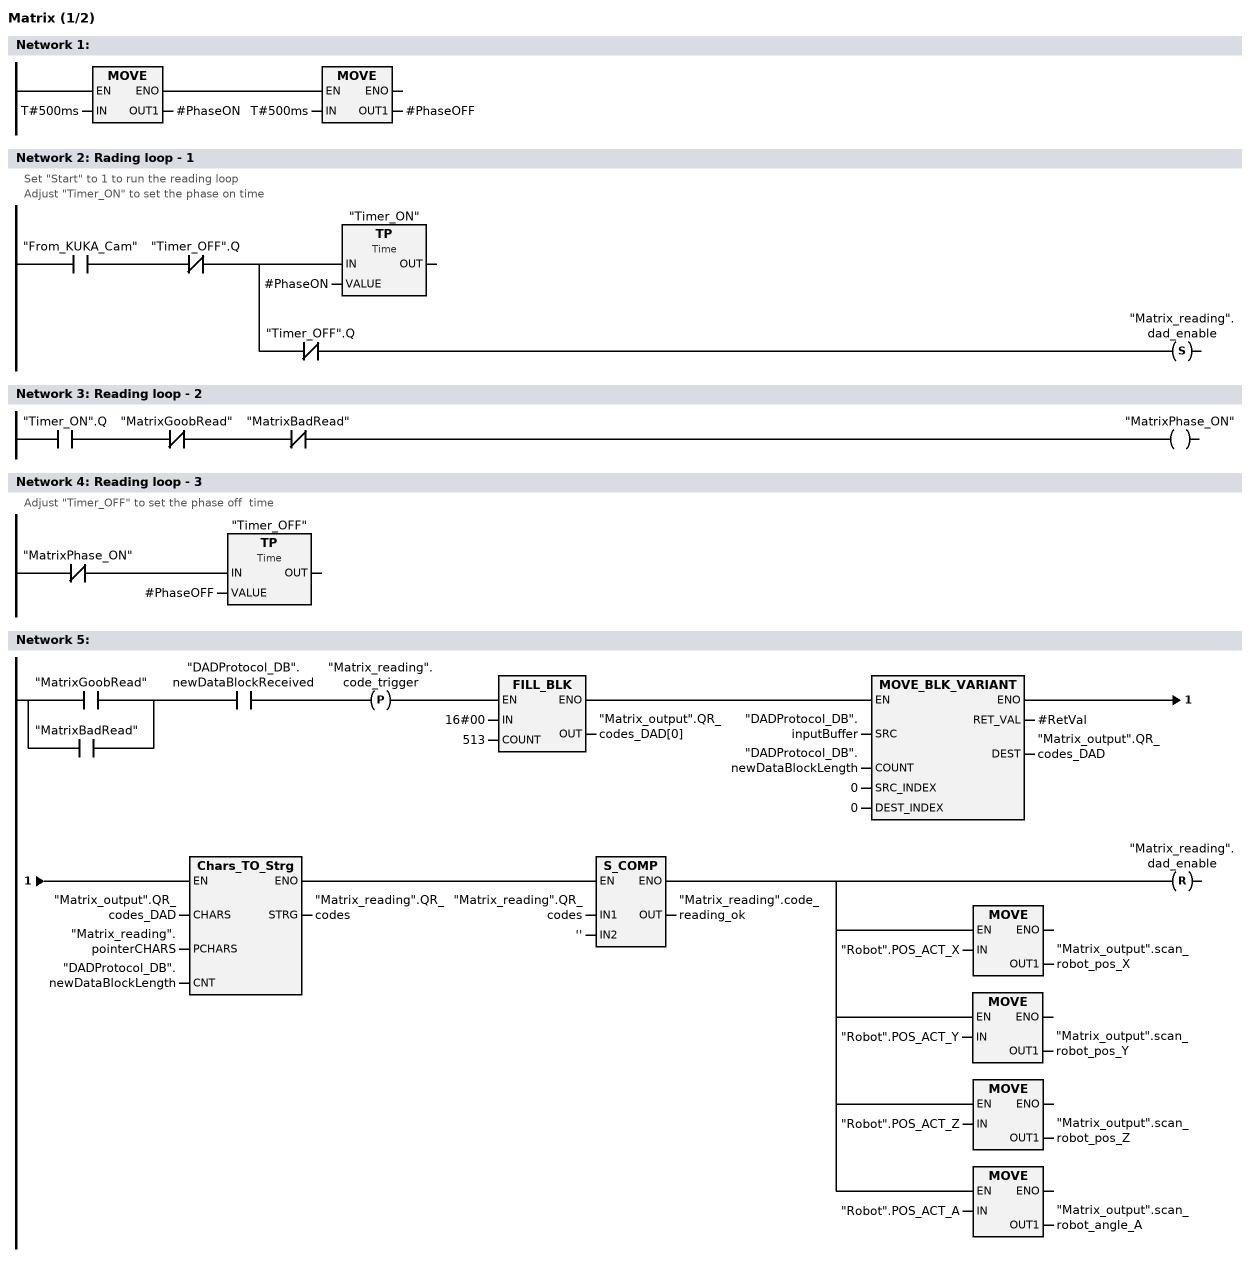
   RUNG wire#powerrail
      { S7_GenerateENO := "TRUE" } Move(in := T#500ms, out1 => #PhaseON)
      { S7_GenerateENO := "TRUE" } Move(in := T#500ms, out1 => #PhaseOFF)
   END_RUNG
   // the same network as SCL:
   // ENO of a box is taken as its EN; it also drops when the box reports an error
   #PhaseON := T#500ms;
   #PhaseOFF := T#500ms;
END_REGION

REGION Network 2: Rading loop - 1
   // Set "Start" to 1 to run the reading loop
   // Adjust "Timer_ON" to set the phase on time
   #_w1 := "From_KUKA_Cam" AND NOT "Timer_OFF".Q;
   "Timer_ON".TP(IN := #_w1, PT := #PhaseON);   // TP coil
   IF #_w1 AND NOT "Timer_OFF".Q THEN "Matrix_reading".dad_enable := TRUE; END_IF;
END_REGION

REGION Network 3: Reading loop - 2
   RUNG wire#powerrail
      Contact( "Timer_ON".Q )
      I_Contact( "MatrixGoobRead" )
      I_Contact( "MatrixBadRead" )
      Coil( "MatrixPhase_ON" )
   END_RUNG
   // the same network as SCL:
   "MatrixPhase_ON" := "Timer_ON".Q AND NOT "MatrixGoobRead" AND NOT "MatrixBadRead";
END_REGION

REGION Network 4: Reading loop - 3
   // Adjust "Timer_OFF" to set the phase off  time
   "Timer_OFF".TP(IN := NOT "MatrixPhase_ON", PT := #PhaseOFF);   // TP coil
END_REGION

REGION Network 5
   // no SCL statement known for Chars_TO_Strg: written as a call
   // ENO of a box is taken as its EN; it also drops when the box reports an error
   #_w1 := ("MatrixGoobRead" OR "MatrixBadRead") AND "DADProtocol_DB".newDataBlockReceived;
   #_w2 := #_w1 AND NOT "Matrix_reading".code_trigger;   // rising edge
   "Matrix_reading".code_trigger := #_w1;
   IF #_w2 THEN
       FILL_BLK(IN := 16#00, COUNT := 513, OUT => "Matrix_output".QR_codes_DAD[0]);
       #RetVal := MOVE_BLK_VARIANT(SRC := "DADProtocol_DB".inputBuffer,
                               COUNT := "DADProtocol_DB".newDataBlockLength,
                               SRC_INDEX := 0,
                               DEST_INDEX := 0,
                               DEST => "Matrix_output".QR_codes_DAD);
       Chars_TO_Strg(Chars := "Matrix_output".QR_codes_DAD,
                     pChars := "Matrix_reading".pointerCHARS,
                     Cnt := "DADProtocol_DB".newDataBlockLength,
                     Strg => "Matrix_reading".QR_codes);
       S_COMP(IN1 := "Matrix_reading".QR_codes, IN2 := '', OUT => "Matrix_reading".code_reading_ok);
       "Matrix_reading".dad_enable := FALSE;
       "Matrix_output".scan_robot_pos_X := "Robot".POS_ACT_X;
       "Matrix_output".scan_robot_pos_Y := "Robot".POS_ACT_Y;
       "Matrix_output".scan_robot_pos_Z := "Robot".POS_ACT_Z;
       "Matrix_output".scan_robot_angle_A := "Robot".POS_ACT_A;
   END_IF;
END_REGION

REGION Network 6
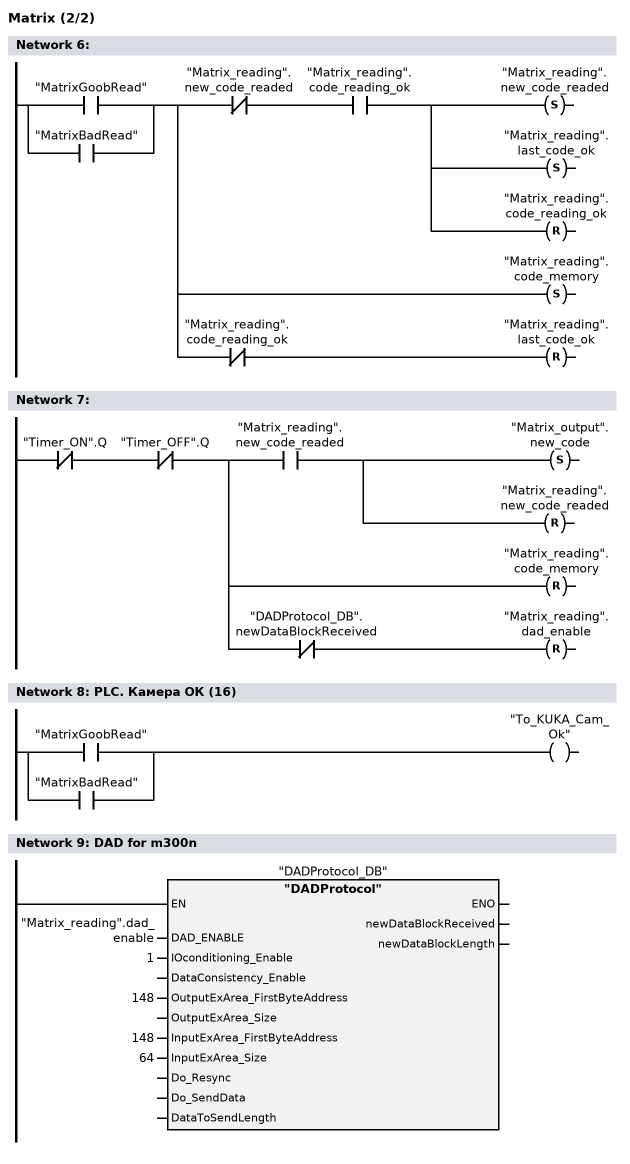
   RUNG wire#powerrail
      Contact( "MatrixGoobRead" )
      wire#w1
      I_Contact( "Matrix_reading".new_code_readed )
      Contact( "Matrix_reading".code_reading_ok )
      wire#w2
      S_Coil( "Matrix_reading".new_code_readed )
   END_RUNG
   RUNG wire#powerrail
      Contact( "MatrixBadRead" )
   END_RUNG wire#w1
   RUNG wire#w2
      S_Coil( "Matrix_reading".last_code_ok )
   END_RUNG
   RUNG wire#w2
      R_Coil( "Matrix_reading".code_reading_ok )
   END_RUNG
   RUNG wire#w1
      S_Coil( "Matrix_reading".code_memory )
   END_RUNG
   RUNG wire#w1
      I_Contact( "Matrix_reading".code_reading_ok )
      R_Coil( "Matrix_reading".last_code_ok )
   END_RUNG
   // the same network as SCL:
   #_w1 := "MatrixGoobRead" OR "MatrixBadRead";
   #_w2 := #_w1 AND NOT "Matrix_reading".new_code_readed AND "Matrix_reading".code_reading_ok;
   IF #_w2 THEN
       "Matrix_reading".new_code_readed := TRUE;
       "Matrix_reading".last_code_ok := TRUE;
       "Matrix_reading".code_reading_ok := FALSE;
   END_IF;
   IF #_w1 THEN "Matrix_reading".code_memory := TRUE; END_IF;
   IF #_w1 AND NOT "Matrix_reading".code_reading_ok THEN "Matrix_reading".last_code_ok := FALSE; END_IF;
END_REGION

REGION Network 7
   RUNG wire#powerrail
      I_Contact( "Timer_ON".Q )
      I_Contact( "Timer_OFF".Q )
      wire#w1
      Contact( "Matrix_reading".new_code_readed )
      wire#w2
      S_Coil( "Matrix_output".new_code )
   END_RUNG
   RUNG wire#w2
      R_Coil( "Matrix_reading".new_code_readed )
   END_RUNG
   RUNG wire#w1
      R_Coil( "Matrix_reading".code_memory )
   END_RUNG
   RUNG wire#w1
      I_Contact( "DADProtocol_DB".newDataBlockReceived )
      R_Coil( "Matrix_reading".dad_enable )
   END_RUNG
   // the same network as SCL:
   #_w1 := NOT "Timer_ON".Q AND NOT "Timer_OFF".Q;
   IF #_w1 AND "Matrix_reading".new_code_readed THEN
       "Matrix_output".new_code := TRUE;
       "Matrix_reading".new_code_readed := FALSE;
   END_IF;
   IF #_w1 THEN "Matrix_reading".code_memory := FALSE; END_IF;
   IF #_w1 AND NOT "DADProtocol_DB".newDataBlockReceived THEN "Matrix_reading".dad_enable := FALSE; END_IF;
END_REGION

REGION Network 8: PLC. Камера ОК (16)
   RUNG wire#powerrail
      Contact( "MatrixGoobRead" )
      wire#w1
      Coil( "To_KUKA_Cam_Ok" )
   END_RUNG
   RUNG wire#powerrail
      Contact( "MatrixBadRead" )
   END_RUNG wire#w1
   // the same network as SCL:
   "To_KUKA_Cam_Ok" := "MatrixGoobRead" OR "MatrixBadRead";
END_REGION

REGION Network 9: DAD for m300n
   RUNG wire#powerrail
      "DADProtocol_DB"(DAD_ENABLE := "Matrix_reading".dad_enable, IOconditioning_Enable := 1, DataConsistency_Enable :=, OutputExArea_FirstByteAddress := 148, OutputExArea_Size :=, InputExArea_FirstByteAddress := 148, InputExArea_Size := 64, Do_Resync :=, Do_SendData :=, DataToSendLength :=, newDataBlockReceived =>, newDataBlockLength =>)
   END_RUNG
   // the same network as SCL:
   "DADProtocol_DB"(DAD_ENABLE := "Matrix_reading".dad_enable,   // "DADProtocol"
                    IOconditioning_Enable := 1,
                    OutputExArea_FirstByteAddress := 148,
                    InputExArea_FirstByteAddress := 148,
                    InputExArea_Size := 64);
END_REGION

REGION Network 11: Reading loop
END_REGION
END_FUNCTION

// folder: 6_OPC

FUNCTION "VC_Proxy" : Void   // FC3, SCL
{ S7_Optimized_Access := 'TRUE' }
VERSION : 0.1
BEGIN
   "To_VC_Rangefinder" := ROR(IN := "To_KUKA_Rangefinder", N := 8);
   "To_VC_Gercon" := "To_KUKA_Gercon";
   "To_VC_PLC_STOP" := "To_KUKA_PLC_STOP";
   "To_VC_PAUSE_STOP" := "To_KUKA_PAUSE_STOP";
   "To_VC_MOVE_ENABLE_KRC" := "To_KUKA_MOVE_ENABLE_KRC";
   "To_VC_PGNO_KRC" := ROR(IN := "To_KUKA_PGNO_KRC", N := 8);
   "To_VC_PGNO_VALID_KRC" := "To_KUKA_PGNO_VALID_KRC";
   "To_VC_PGNO_PARITY" := "To_KUKA_PGNO_PARITY";
   "To_VC_CONF_MESS" := "To_KUKA_CONF_MESS";
   "To_VC_DRIVERS_OFF" := "To_KUKA_DRIVERS_OFF";
   "To_VC_DRIVERS_ON" := "To_KUKA_DRIVERS_ON";
   "To_VC_Collision" := "To_KUKA_Collision";
   "To_VC_QRcode_X" := ROR(IN := "To_KUKA_QRcode_X", N := 8);
   "To_VC_QRcode_Angle" := ROR(IN := "To_KUKA_QRcode_Angle", N := 8);
   "To_VC_EXT_START_KRC" := "To_KUKA_EXT_START_KRC";
   "To_VC_Vacuum_Ok" := "To_KUKA_Vacuum_Ok";
   "To_VC_QRcode_Y" := ROR(IN := "To_KUKA_QRcode_Y", N := 8);
   "To_VC_Cam_Ok" := "To_KUKA_Cam_Ok";
   "To_VC_IsGripperMainHome" := "To_KUKA_IsGripperMainHome";
   "To_VC_IsGripperFeederHome" := "To_KUKA_IsGripperFeederHome";
   "To_VC_Part_length_X" := ROR(IN := "To_KUKA_Part_length_X", N := 8);
   "To_VC_Part_thickness_Z" := ROR(IN := "To_KUKA_Part_thickness_Z", N := 8);
   "To_VC_GripperRetracted" := "To_KUKA_GripperRetracted";
   "To_VC_PartEndSwitch_1" := "To_KUKA_PartEndSwitch_1";
   "To_VC_PartEndSwitch_2" := "To_KUKA_PartEndSwitch_2";
   "To_VC_Gripper_Sign_X" := "To_KUKA_Gripper_Sign_X";
   "To_VC_Gripper_Sign_Y" := "To_KUKA_Gripper_Sign_Y";
   "To_VC_FlipTableOpened" := "To_KUKA_FlipTableOpened";
   "To_VC_FlipTableClosed" := "To_KUKA_FlipTableClosed";
   "To_VC_Part_length_Y" := ROR(IN := "To_KUKA_Part_length_Y", N := 8);
   "To_VC_QRcode_Z" := ROR(IN := "To_KUKA_QRcode_Z", N := 8);
   "To_VC_Part_X" := ROR(IN := "To_KUKA_Part_X", N := 8);
   "To_VC_Part_Y" := ROR(IN := "To_KUKA_Part_Y", N := 8);
   "To_VC_Part_A" := ROR(IN := "To_KUKA_Part_A", N := 8);
   "To_VC_Part_Z" := ROR(IN := "To_KUKA_Part_Z", N := 8);
   "To_VC_Part_Length_X0" := ROR(IN := "To_KUKA_Part_Length_X0", N := 8);
   "To_VC_Part_Length_Y0" := ROR(IN := "To_KUKA_Part_Length_Y0", N := 8);
   "To_VC_Gripper_Within_part" := "To_KUKA_Gripper_Within_part";
   "To_VC_Part_Slot" := ROR(IN := "To_KUKA_Part_Slot", N := 8);
   "To_VC_Free_Slot" := ROR(IN := "To_KUKA_Free_Slot", N := 8);
   "To_VC_AckPalletScanned" := "To_KUKA_AckPalletScanned";
   "To_VC_Slot_X" := ROR(IN := "To_KUKA_Slot_X", N := 8);
   "To_VC_Slot_Y" := ROR(IN := "To_KUKA_Slot_Y", N := 8);
   "To_VC_Slot_Z" := ROR(IN := "To_KUKA_Slot_Z", N := 8);
   "To_VC_Slot_A" := ROR(IN := "To_KUKA_Slot_A", N := 8);
   "To_VC_WithoutMachine" := "To_KUKA_WithoutMachine";
   "To_VC_Part_Destination" := ROR(IN := "To_KUKA_Part_Destination", N := 8);


   "Robot"."ALARM_STOP_KRC":="From_VC_ALARM_STOP_KRC";
   "Robot"."FlipVacuumOn" := "From_VC_FlipVacuumOn";
   "Robot"."Pallet_Scanned" := "From_VC_Pallet_Scanned";
   "Robot"."ERROR_KRC" := "From_VC_ERROR_KRC";
   "Robot"."PRO_ACT_KRC" := "From_VC_PRO_ACT_KRC";
   "Robot"."PartMeasuring" := "From_VC_PartMeasuring";
   "Robot"."PartOK" := "From_VC_PartOK";
   "Robot"."SetFlipClose" := "From_VC_SetFlipClose";
   "Robot"."Flow2PartON" := "From_VC_Flow2PartON";
   "Robot"."SetRetract" := "From_VC_SetRetract";
   "Robot"."SetPressureOFF" := "From_VC_SetPressureOFF";
   "Robot"."EXT_FIRST_START" := "From_VC_EXT_FIRST_START";
   "Robot"."LifeBit" := "From_VC_LifeBit";
   "Robot"."SetVacuumON" := "From_VC_SetVacuumON";
   "Robot"."APPL_RUN_KRC" := "From_VC_APPL_RUN_KRC";
   "Robot"."EXT_ACTIVE" := "From_VC_EXT_ACTIVE";
   "Robot"."PERI_RDY_KRC" := "From_VC_PERI_RDY_KRC";
   "Robot"."STOPMESS_KRC" := "From_VC_STOPMESS_KRC";
   "Robot"."Cam" := "From_VC_Cam";
   "Robot"."PRO_MOVE_KRC" := "From_VC_PRO_MOVE_KRC";
   "Robot"."IN_HOME_KRC" := "From_VC_IN_HOME_KRC";
   "Robot"."USER_SAF_KRC" := "From_VC_USER_SAF_KRC";
   "Robot"."ROB_CAL_KRC" := "From_VC_ROB_CAL_KRC";
   "Robot"."I_O_ACTCONF_KRC" := "From_VC_I_O_ACTCONF_KRC";
   "Robot"."RC_RDY1_KRC" := "From_VC_RC_RDY1_KRC";
   "Robot"."PGNO_REQ_KRC" := "From_VC_PGNO_REQ_KRC";
   "Robot"."PGNO_REFL_KRC" := ROR(IN := "From_VC_PGNO_REFL_KRC", N := 8);
   //"Robot"."AXIS_ACT_A1" := ROR(IN := "From_VC_AXIS_ACT_A1", N := 8);
   //"Robot"."POS_ACT_Z" := ROR(IN := "From_VC_POS_ACT_Z", N := 8);
   //"Robot"."POS_ACT_Y" := ROR(IN := "From_VC_POS_ACT_Y", N := 8);
   //"Robot"."POS_ACT_X" := ROR(IN := "From_VC_POS_ACT_X", N := 8);
   //"Robot"."POS_ACT_A" := ROR(IN := "From_VC_POS_ACT_A", N := 8);
   "Robot"."Part_Status" := ROR(IN := "From_VC_Part_Status", N := 8);
   "Robot"."Serial_Number" := ROR(IN := "From_VC_Serial_Number", N := 8);


   "Get_IN"(In_val := "From_KUKA_AXIS_ACT_A1",
            Out_val := "Robot".AXIS_ACT_A1);
   "Get_IN"(In_val := "From_KUKA_POS_ACT_X",
            Out_val := "Robot".POS_ACT_X);
   "Get_IN"(In_val := "From_KUKA_POS_ACT_Y",
            Out_val := "Robot".POS_ACT_Y);
   "Get_IN"(In_val := "From_KUKA_POS_ACT_Z",
            Out_val := "Robot".POS_ACT_Z);
   "Get_IN"(In_val := "From_KUKA_POS_ACT_A",
            Out_val := "Robot".POS_ACT_A);

   "To_VC_IsGripperMainHome" := NOT "From_VC_SetRetract" AND NOT "From_VC_SetPressureOFF";
   "To_VC_Cam_Ok" := "From_KUKA_Cam";
   "To_VC_Test_DInt" := -15;
END_FUNCTION

FUNCTION "PROFINET_Proxy" : Void   // FC4, SCL
{ S7_Optimized_Access := 'TRUE' }
VERSION : 0.1
BEGIN
   "Robot"."ALARM_STOP_KRC":="From_KUKA_ALARM_STOP_KRC";
   "Robot"."FlipVacuumOn" := "From_KUKA_FlipVacuumOn";
   "Robot"."Pallet_Scanned" := "From_KUKA_Pallet_Scanned";
   "Robot"."ERROR_KRC" := "From_KUKA_ERROR_KRC";
   "Robot"."PRO_ACT_KRC" := "From_KUKA_PRO_ACT_KRC";
   "Robot"."PartMeasuring" := "From_KUKA_PartMeasuring";
   "Robot"."PartOK" := "From_KUKA_PartOK";
   "Robot"."SetFlipClose" := "From_KUKA_SetFlipClose";
   "Robot"."Flow2PartON" := "From_KUKA_Flow2PartON";
   "Robot"."SetRetract" := "From_KUKA_SetRetract";
   "Robot"."SetPressureOFF" := "From_KUKA_SetPressureOFF";
   "Robot"."EXT_FIRST_START" := "From_KUKA_EXT_FIRST_START";
   "Robot"."LifeBit" := "From_KUKA_LifeBit";
   "Robot"."SetVacuumON" := "From_KUKA_SetVacuumON";
   "Robot"."APPL_RUN_KRC" := "From_KUKA_APPL_RUN_KRC";
   "Robot"."EXT_ACTIVE" := "From_KUKA_EXT_ACTIVE";
   "Robot"."PERI_RDY_KRC" := "From_KUKA_PERI_RDY_KRC";
   "Robot"."STOPMESS_KRC" := "From_KUKA_STOPMESS_KRC";
   "Robot"."Cam" := "From_KUKA_Cam";
   "Robot"."PRO_MOVE_KRC" := "From_KUKA_PRO_MOVE_KRC";
   "Robot"."IN_HOME_KRC" := "From_KUKA_IN_HOME_KRC";
   "Robot"."USER_SAF_KRC" := "From_KUKA_USER_SAF_KRC";
   "Robot"."ROB_CAL_KRC" := "From_KUKA_ROB_CAL_KRC";
   "Robot"."I_O_ACTCONF_KRC" := "From_KUKA_I_O_ACTCONF_KRC";
   "Robot"."RC_RDY1_KRC" := "From_KUKA_RC_RDY1_KRC";
   "Robot"."PGNO_REQ_KRC" := "From_KUKA_PGNO_REQ_KRC"; 
   "Robot"."PGNO_REFL_KRC" := "From_KUKA_PGNO_REFL_KRC"; //no ROR 
   //"Robot"."AXIS_ACT_A1" := ROR(IN := "From_KUKA_AXIS_ACT_A1", N := 8);
   //"Robot"."POS_ACT_Z" := ROR(IN := "From_KUKA_POS_ACT_Z", N := 8);
   //"Robot"."POS_ACT_Y" := ROR(IN := "From_KUKA_POS_ACT_Y", N := 8);
   //"Robot"."POS_ACT_X" := ROR(IN := "From_KUKA_POS_ACT_X", N := 8);
   //"Robot"."POS_ACT_A" := ROR(IN := "From_KUKA_POS_ACT_A", N := 8);
   "Robot"."Part_Status" := ROR(IN := "From_KUKA_Part_Status", N := 8);
   "Robot"."Serial_Number" := ROR(IN := "From_KUKA_Serial_Number", N := 8);

   "Get_IN"(In_val := "From_KUKA_AXIS_ACT_A1",
            Out_val := "Robot".AXIS_ACT_A1);
   "Get_IN"(In_val := "From_KUKA_POS_ACT_X",
            Out_val := "Robot".POS_ACT_X);
   "Get_IN"(In_val := "From_KUKA_POS_ACT_Y",
            Out_val := "Robot".POS_ACT_Y);
   "Get_IN"(In_val := "From_KUKA_POS_ACT_Z",
            Out_val := "Robot".POS_ACT_Z);
   "Get_IN"(In_val := "From_KUKA_POS_ACT_A",
            Out_val := "Robot".POS_ACT_A);
END_FUNCTION

FUNCTION "ResetJob" : Void   // FC10, SCL
{ S7_Optimized_Access := 'TRUE' }
VERSION : 0.1
   VAR_IN_OUT
      in_Task : "TypeRobotTask";
   END_VAR
BEGIN
           #in_Task.program_fullpath := '';
           #in_Task.part_length_X := 0;
           #in_Task.part_length_Y := 0;
           #in_Task.part_thickness_Z := 0;
           #in_Task.part_pos_X := 0;
           #in_Task.part_pos_Y := 0;
           #in_Task.part_pos_Z := 0;
           #in_Task.part_angle_A := 0;
           #in_Task.operation_side := ' ';
           #in_Task.part_side := ' ';
           #in_Task.lay_number := 0;
           #in_Task.operation_type := '';
           #in_Task.operation_number := 0;
           #in_Task.robot_task_id := 0;
           #in_Task.part_id := 0;
           #in_Task.part_number := 0;
           #in_Task.order_id := 0;
           #in_Task.plc_id := 0;
           #in_Task.machine_status := '';
           #in_Task.robot_status := '';
           #in_Task.task_status := 'finish';
           #in_Task.part_status := 'done';
           #in_Task.plc_ip := '';
           #in_Task.plc_name := '';
           #in_Task.robot_name := '';
           #in_Task.part_length_X0 := 0;
           #in_Task.part_length_Y0 := 0;
           #in_Task.slot_pos_X := 0;
           #in_Task.slot_pos_Y := 0;
           #in_Task.slot_pos_Z := 0;
           #in_Task.slot_angle_A := 0;
           #in_Task.part_slot := 0;
           #in_Task.free_slot := 0;
           //#in_Task.start_job := FALSE;
END_FUNCTION

ORGANIZATION_BLOCK "Startup"   // OB100, LAD, Startup
TITLE = "Complete Restart"
{ S7_Optimized_Access := 'TRUE' }
VERSION : 0.1
   VAR_INPUT
      LostRetentive : Bool;   // True if retentive data are lost
      LostRTC : Bool;   // True if date and time are lost
   END_VAR
BEGIN

REGION Network 1
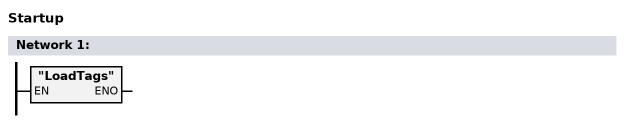
   RUNG wire#powerrail
      "LoadTags"()
   END_RUNG
   // the same network as SCL:
   "LoadTags"();
END_REGION
END_ORGANIZATION_BLOCK

// folder: 7_Tags

FUNCTION "AddTag" : Void   // FC5, SCL
{ S7_Optimized_Access := 'TRUE' }
VERSION : 0.1
   VAR_INPUT
      DB_number : UInt;
      Robot_number : USInt;
      "Name" : String;
      "Type" : String;
      Use : String;
      ReadOnly : USInt;
      OffsetByte : UInt;
      OffsetBit : USInt;
   END_VAR
BEGIN
   "PLC_tags".Tags["PLC_tags".Tags_count].DB_number := #DB_number;
   "PLC_tags".Tags["PLC_tags".Tags_count].Robot_number := #Robot_number;
   "PLC_tags".Tags["PLC_tags".Tags_count].Name := #Name;
   "PLC_tags".Tags["PLC_tags".Tags_count].Type := #Type;
   "PLC_tags".Tags["PLC_tags".Tags_count].Use := #Use;
   "PLC_tags".Tags["PLC_tags".Tags_count].ReadOnly := #ReadOnly;
   "PLC_tags".Tags["PLC_tags".Tags_count].OffsetByte := #OffsetByte;
   "PLC_tags".Tags["PLC_tags".Tags_count].OffsetBit := #OffsetBit;

   "PLC_tags".Tags_count := "PLC_tags".Tags_count + 1;
END_FUNCTION

FUNCTION "LoadTags" : Void   // FC6, SCL
{ S7_Optimized_Access := 'TRUE' }
VERSION : 0.1
BEGIN
   IF "PLC_tags".Tags_count <> 64 THEN

       "PLC_tags".Tags_count := 0;

       "AddTag"(Robot_number := 1,
                Name := 'new_code',
                Type := 'Bool',
                Use := 'InOut',
                ReadOnly := 0,
                DB_number := 10,
                OffsetByte := 0,
                OffsetBit := 0);
       "AddTag"(Robot_number := 1,
                Name := 'scan_robot_pos_x',
                Type := 'Real',
                Use := 'Out',
                ReadOnly := 1,
                DB_number := 10,
                OffsetByte := 2,
                OffsetBit := 0);
       "AddTag"(Robot_number := 1,
                Name := 'scan_robot_pos_y',
                Type := 'Real',
                Use := 'Out',
                ReadOnly := 1,
                DB_number := 10,
                OffsetByte := 6,
                OffsetBit := 0);
       "AddTag"(Robot_number := 1,
                Name := 'scan_robot_pos_z',
                Type := 'Real',
                Use := 'Out',
                ReadOnly := 1,
                DB_number := 10,
                OffsetByte := 10,
                OffsetBit := 0);
       "AddTag"(Robot_number := 1,
                Name := 'scan_robot_angle_a',
                Type := 'Real',
                Use := 'Out',
                ReadOnly := 1,
                DB_number := 10,
                OffsetByte := 14,
                OffsetBit := 0);
       "AddTag"(Robot_number := 1,
                Name := 'scan_lay_number',
                Type := 'USInt',
                Use := 'Out',
                ReadOnly := 0,
                DB_number := 10,
                OffsetByte := 18,
                OffsetBit := 0);
       "AddTag"(Robot_number := 1,
                Name := 'qr_codes_dad',
                Type := 'Array[0..512] of Byte',
                Use := 'Out',
                ReadOnly := 1,
                DB_number := 10,
                OffsetByte := 20,
                OffsetBit := 0);
       "AddTag"(Robot_number := 1,
                Name := 'not_sended2arduino',
                Type := 'Bool',
                Use := 'In',
                ReadOnly := 1,
                DB_number := 1,
                OffsetByte := 0,
                OffsetBit := 0);
       "AddTag"(Robot_number := 1,
                Name := 'not_sended2bhx',
                Type := 'Bool',
                Use := 'In',
                ReadOnly := 0,
                DB_number := 1,
                OffsetByte := 0,
                OffsetBit := 1);
       "AddTag"(Robot_number := 1,
                Name := 'new_part',
                Type := 'Bool',
                Use := 'In',
                ReadOnly := 0,
                DB_number := 1,
                OffsetByte := 0,
                OffsetBit := 2);
       "AddTag"(Robot_number := 1,
                Name := 'start_job',
                Type := 'Bool',
                Use := 'In',
                ReadOnly := 0,
                DB_number := 1,
                OffsetByte := 0,
                OffsetBit := 3);
       "AddTag"(Robot_number := 1,
                Name := 'reset_job',
                Type := 'Bool',
                Use := 'In',
                ReadOnly := 0,
                DB_number := 1,
                OffsetByte := 0,
                OffsetBit := 4);
       "AddTag"(Robot_number := 1,
                Name := 'robot_alarm_reset',
                Type := 'Bool',
                Use := 'In',
                ReadOnly := 0,
                DB_number := 1,
                OffsetByte := 0,
                OffsetBit := 5);
       "AddTag"(Robot_number := 1,
                Name := 'w/o_machine_mode',
                Type := 'Bool',
                Use := 'In',
                ReadOnly := 0,
                DB_number := 1,
                OffsetByte := 0,
                OffsetBit := 6);
       "AddTag"(Robot_number := 1,
                Name := 'gripper_sign_x',
                Type := 'Bool',
                Use := 'In',
                ReadOnly := 0,
                DB_number := 1,
                OffsetByte := 0,
                OffsetBit := 7);
       "AddTag"(Robot_number := 1,
                Name := 'gripper_sign_y',
                Type := 'Bool',
                Use := 'In',
                ReadOnly := 0,
                DB_number := 1,
                OffsetByte := 1,
                OffsetBit := 0);
       "AddTag"(Robot_number := 1,
                Name := 'gripper_within_part',
                Type := 'Bool',
                Use := 'In',
                ReadOnly := 0,
                DB_number := 1,
                OffsetByte := 1,
                OffsetBit := 1);
       "AddTag"(Robot_number := 1,
                Name := 'robot_pause',
                Type := 'Bool',
                Use := 'In',
                ReadOnly := 0,
                DB_number := 1,
                OffsetByte := 1,
                OffsetBit := 2);
       "AddTag"(Robot_number := 1,
                Name := 'pallet_scanned',
                Type := 'Bool',
                Use := 'In',
                ReadOnly := 0,
                DB_number := 1,
                OffsetByte := 1,
                OffsetBit := 3);
       "AddTag"(Robot_number := 1,
                Name := 'new_pallet',
                Type := 'Bool',
                Use := 'In',
                ReadOnly := 0,
                DB_number := 1,
                OffsetByte := 1,
                OffsetBit := 4);
       "AddTag"(Robot_number := 1,
                Name := 'robot_in_home',
                Type := 'Bool',
                Use := 'In',
                ReadOnly := 1,
                DB_number := 1,
                OffsetByte := 1,
                OffsetBit := 5);
       "AddTag"(Robot_number := 1,
                Name := 'program_fullpath',
                Type := 'String[99]',
                Use := 'In',
                ReadOnly := 0,
                DB_number := 1,
                OffsetByte := 2,
                OffsetBit := 0);
       "AddTag"(Robot_number := 1,
                Name := 'part_length_x',
                Type := 'UInt',
                Use := 'In',
                ReadOnly := 0,
                DB_number := 1,
                OffsetByte := 104,
                OffsetBit := 0);
       "AddTag"(Robot_number := 1,
                Name := 'part_length_y',
                Type := 'UInt',
                Use := 'In',
                ReadOnly := 0,
                DB_number := 1,
                OffsetByte := 106,
                OffsetBit := 0);
       "AddTag"(Robot_number := 1,
                Name := 'part_thickness_z',
                Type := 'UInt',
                Use := 'In',
                ReadOnly := 0,
                DB_number := 1,
                OffsetByte := 108,
                OffsetBit := 0);
       "AddTag"(Robot_number := 1,
                Name := 'part_pos_x',
                Type := 'Real',
                Use := 'InOut',
                ReadOnly := 0,
                DB_number := 1,
                OffsetByte := 110,
                OffsetBit := 0);
       "AddTag"(Robot_number := 1,
                Name := 'part_pos_y',
                Type := 'Real',
                Use := 'InOut',
                ReadOnly := 0,
                DB_number := 1,
                OffsetByte := 114,
                OffsetBit := 0);
       "AddTag"(Robot_number := 1,
                Name := 'part_pos_z',
                Type := 'Real',
                Use := 'InOut',
                ReadOnly := 0,
                DB_number := 1,
                OffsetByte := 118,
                OffsetBit := 0);
       "AddTag"(Robot_number := 1,
                Name := 'part_angle_a',
                Type := 'Real',
                Use := 'InOut',
                ReadOnly := 0,
                DB_number := 1,
                OffsetByte := 122,
                OffsetBit := 0);
       "AddTag"(Robot_number := 1,
                Name := 'part_side',
                Type := 'Char',
                Use := 'In',
                ReadOnly := 0,
                DB_number := 1,
                OffsetByte := 126,
                OffsetBit := 0);
       "AddTag"(Robot_number := 1,
                Name := 'part_slot',
                Type := 'USInt',
                Use := 'In',
                ReadOnly := 1,
                DB_number := 1,
                OffsetByte := 127,
                OffsetBit := 0);
       "AddTag"(Robot_number := 1,
                Name := 'free_slot',
                Type := 'USInt',
                Use := 'In',
                ReadOnly := 1,
                DB_number := 1,
                OffsetByte := 128,
                OffsetBit := 0);
       "AddTag"(Robot_number := 1,
                Name := 'operation_side',
                Type := 'Char',
                Use := 'In',
                ReadOnly := 1,
                DB_number := 1,
                OffsetByte := 129,
                OffsetBit := 0);
       "AddTag"(Robot_number := 1,
                Name := 'operation_number',
                Type := 'Int',
                Use := 'In',
                ReadOnly := 1,
                DB_number := 1,
                OffsetByte := 130,
                OffsetBit := 0);
       "AddTag"(Robot_number := 1,
                Name := 'lay_number',
                Type := 'Int',
                Use := 'In',
                ReadOnly := 1,
                DB_number := 1,
                OffsetByte := 132,
                OffsetBit := 0);
       "AddTag"(Robot_number := 1,
                Name := 'robot_task_id',
                Type := 'LInt',
                Use := 'In',
                ReadOnly := 1,
                DB_number := 1,
                OffsetByte := 134,
                OffsetBit := 0);
       "AddTag"(Robot_number := 1,
                Name := 'robot_id',
                Type := 'LInt',
                Use := 'In',
                ReadOnly := 1,
                DB_number := 1,
                OffsetByte := 142,
                OffsetBit := 0);
       "AddTag"(Robot_number := 1,
                Name := 'part_id',
                Type := 'LInt',
                Use := 'In',
                ReadOnly := 1,
                DB_number := 1,
                OffsetByte := 150,
                OffsetBit := 0);
       "AddTag"(Robot_number := 1,
                Name := 'part_number',
                Type := 'LInt',
                Use := 'In',
                ReadOnly := 1,
                DB_number := 1,
                OffsetByte := 158,
                OffsetBit := 0);
       "AddTag"(Robot_number := 1,
                Name := 'order_id',
                Type := 'LInt',
                Use := 'In',
                ReadOnly := 1,
                DB_number := 1,
                OffsetByte := 166,
                OffsetBit := 0);
       "AddTag"(Robot_number := 0,
                Name := 'plc_id',
                Type := 'LInt',
                Use := 'In',
                ReadOnly := 1,
                DB_number := 1,
                OffsetByte := 174,
                OffsetBit := 0);
       "AddTag"(Robot_number := 1,
                Name := 'robot_program',
                Type := 'UInt',
                Use := 'In',
                ReadOnly := 1,
                DB_number := 1,
                OffsetByte := 182,
                OffsetBit := 0);
       "AddTag"(Robot_number := 1,
                Name := 'operation_type',
                Type := 'String[30]',
                Use := 'In',
                ReadOnly := 1,
                DB_number := 1,
                OffsetByte := 184,
                OffsetBit := 0);
       "AddTag"(Robot_number := 1,
                Name := 'machine_status',
                Type := 'String[30]',
                Use := 'Out',
                ReadOnly := 1,
                DB_number := 1,
                OffsetByte := 216,
                OffsetBit := 0);
       "AddTag"(Robot_number := 1,
                Name := 'robot_trajectory',
                Type := 'String[30]',
                Use := 'Out',
                ReadOnly := 1,
                DB_number := 1,
                OffsetByte := 248,
                OffsetBit := 0);
       "AddTag"(Robot_number := 1,
                Name := 'robot_status',
                Type := 'String[30]',
                Use := 'Out',
                ReadOnly := 1,
                DB_number := 1,
                OffsetByte := 280,
                OffsetBit := 0);
       "AddTag"(Robot_number := 1,
                Name := 'task_status',
                Type := 'String[30]',
                Use := 'InOut',
                ReadOnly := 0,
                DB_number := 1,
                OffsetByte := 312,
                OffsetBit := 0);
       "AddTag"(Robot_number := 1,
                Name := 'part_status',
                Type := 'String[30]',
                Use := 'InOut',
                ReadOnly := 0,
                DB_number := 1,
                OffsetByte := 344,
                OffsetBit := 0);
       "AddTag"(Robot_number := 1,
                Name := 'part_source',
                Type := 'String[30]',
                Use := 'In',
                ReadOnly := 0,
                DB_number := 1,
                OffsetByte := 376,
                OffsetBit := 0);
       "AddTag"(Robot_number := 1,
                Name := 'part_destination',
                Type := 'String[30]',
                Use := 'In',
                ReadOnly := 0,
                DB_number := 1,
                OffsetByte := 408,
                OffsetBit := 0);
       "AddTag"(Robot_number := 0,
                Name := 'plc_ip',
                Type := 'String[30]',
                Use := 'In',
                ReadOnly := 0,
                DB_number := 1,
                OffsetByte := 440,
                OffsetBit := 0);
       "AddTag"(Robot_number := 0,
                Name := 'plc_name',
                Type := 'String[30]',
                Use := 'In',
                ReadOnly := 0,
                DB_number := 1,
                OffsetByte := 472,
                OffsetBit := 0);
       "AddTag"(Robot_number := 1,
                Name := 'robot_name',
                Type := 'String[30]',
                Use := 'In',
                ReadOnly := 0,
                DB_number := 1,
                OffsetByte := 504,
                OffsetBit := 0);
       "AddTag"(Robot_number := 1,
                Name := 'part_length_x0',
                Type := 'UInt',
                Use := 'In',
                ReadOnly := 0,
                DB_number := 1,
                OffsetByte := 536,
                OffsetBit := 0);
       "AddTag"(Robot_number := 1,
                Name := 'part_length_y0',
                Type := 'UInt',
                Use := 'In',
                ReadOnly := 0,
                DB_number := 1,
                OffsetByte := 538,
                OffsetBit := 0);
       "AddTag"(Robot_number := 1,
                Name := 'slot_pos_x',
                Type := 'Real',
                Use := 'InOut',
                ReadOnly := 0,
                DB_number := 1,
                OffsetByte := 540,
                OffsetBit := 0);
       "AddTag"(Robot_number := 1,
                Name := 'slot_pos_y',
                Type := 'Real',
                Use := 'InOut',
                ReadOnly := 0,
                DB_number := 1,
                OffsetByte := 544,
                OffsetBit := 0);
       "AddTag"(Robot_number := 1,
                Name := 'slot_pos_z',
                Type := 'Real',
                Use := 'InOut',
                ReadOnly := 0,
                DB_number := 1,
                OffsetByte := 548,
                OffsetBit := 0);
       "AddTag"(Robot_number := 1,
                Name := 'slot_angle_a',
                Type := 'Real',
                Use := 'InOut',
                ReadOnly := 0,
                DB_number := 1,
                OffsetByte := 552,
                OffsetBit := 0);
       "AddTag"(Robot_number := 1,
                Name := 'out_pos_x',
                Type := 'Real',
                Use := 'In',
                ReadOnly := 0,
                DB_number := 1,
                OffsetByte := 556,
                OffsetBit := 0);
       "AddTag"(Robot_number := 1,
                Name := 'out_pos_y',
                Type := 'Real',
                Use := 'In',
                ReadOnly := 0,
                DB_number := 1,
                OffsetByte := 560,
                OffsetBit := 0);
       "AddTag"(Robot_number := 1,
                Name := 'out_pos_z',
                Type := 'Real',
                Use := 'In',
                ReadOnly := 0,
                DB_number := 1,
                OffsetByte := 564,
                OffsetBit := 0);
       "AddTag"(Robot_number := 1,
                Name := 'out_pos_a',
                Type := 'Real',
                Use := 'In',
                ReadOnly := 0,
                DB_number := 1,
                OffsetByte := 568,
                OffsetBit := 0);
       "AddTag"(Robot_number := 1,
                Name := 'robot_serial',
                Type := 'UInt',
                Use := 'In',
                ReadOnly := 0,
                DB_number := 1,
                OffsetByte := 572,
                OffsetBit := 0);
       "AddTag"(Robot_number := 1,
                Name := 'Test_DInt',
                Type := 'DInt',
                Use := 'Out',
                ReadOnly := 0,
                DB_number := 1,
                OffsetByte := 574,
                OffsetBit := 0);
   END_IF;
END_FUNCTION

// ===== library types =====

// folder: LGF/1 Date and timer operations

FUNCTION "LGF_GetCalendarDay" : DInt   // FC10028, SCL
TITLE = LGF_GetCalendarDay
{ S7_Optimized_Access := 'TRUE' }
AUTHOR : Siemens_Digital_Industry
FAMILY : LGF
NAME : LGF_GetCalendarDay
// This function uses the specified date to calculate the number of days that have passed since the beginning of the year (1st January).
// 
// The function is used in the functions “LGF_GetCalendarWeek_ISO” and “LGF_GetCalendarWeek_US”.
// Diese Funktion berechnet aus dem vorgegebenen Datum die Anzahl der Tage, die seit dem Anfang des Jahres vergangen sind (1. Januar).
// 
// Die Funktion wird in den Funktionen "LGF_GetCalendarWeek_ISO" und "LGF_GetCalendarWeek_US" verwendet.
   VAR_INPUT
      "date" : DTL;   // Date for the calculation of the calendar days since 1 January. / Datum für die Berechnung der vergangenen Kalendertagen seit dem 01. Januar
   END_VAR
   VAR_OUTPUT
      error : Bool;   // FALSE: No error / TRUE: An error occurred during the execution of the FB / FALSE: Kein Fehler / TRUE: Während der Ausführung des FB ist ein Fehler aufgetreten
      status : Word;   // 16#0000-16#7FFF: Status of the FB / 16#8000-16#FFFF: Error identification (see following Table) / 16#0000-16#7FFF: Status des FB / 16#8000-16#FFFF: Fehleridentifikation (siehe folgende Tabelle)
   END_VAR
   VAR_TEMP
      tempDaysPassed : DInt;   // Temp tag for the number of days past / Temp Variable für die Anzahl der vergangenen Tage
      tempDate : DTL;   // Temp variable to store date for calculations / Temp Variable um Datum für Berechung zwischen zu speichern
   END_VAR
   // Ret_Val : Days past since January 1st. / Vergangene Tage seit 1. Januar.
   VAR CONSTANT
      FIRST_DAY : USInt := 1;   // 1st of a month / 1. Tag eines Monats
      LAST_DAY : USInt := 31;   // 31st of a month / 31. Tag eines Monats
      JANUARY : USInt := 1;   // Month number for January / Monatsnumer Januar
      DECEMBER : USInt := 12;   // Month number for December / Monatsnummer Dezember
      TIME_ZERO_FORCE_UPDATE : Time := t#0d;   // By adding zero an update of DTL Tag is forced and auto checks are applied / Durch die Addition von "0" wird ein Update üder den Zeitstemple erstellt und ebenfalls auf gültigkeit geprüft.
      ONE_DAY : DInt := 1;   // One single day for incrementing / Ein Tag für inkrementierungen
      STATUS_NO_ERROR : Word := 16#0000;   // Status: no error occurred / Status: kein Fehler aufgetreten
      ERR_LIM_DATE : Word := 16#8201;   // Date out of the range, has to be greater than <1970-01-01 ; 2262-04-11> / Datum ausserhalb des gültigen Bereiches, es muss nach dem <1970-01-01 ; 2262-04-11> liegen
   END_VAR
BEGIN
   REGION BLOCK INFO HEADER
     //===============================================================================
     // SIEMENS AG / (c)Copyright 2019
     //-------------------------------------------------------------------------------
     // Title:            LGF_GetCalendarDay
     // Comment/Function: This function calculates for a date the passed days since 1st January.
     // Library/Family:   LGF(Library General Functions)
     // Author:           Siemens Digital Industry Support
     // Tested with:      S7-PLCSIM Advanced V2.0 SP1
     // Engineering:      TIA Portal V15.1
     // Restrictions:     ENO disabled - error handling done with error and status
     // Requirements:     PLC (S7-1200 / S7-1500)
     //-------------------------------------------------------------------------------
     // Change log table:
     // Version  | Date       | Expert in charge       | Changes applied
     //----------|------------|------------------------|------------------------------
     // 01.00.00 16.07.2019  Simatic Systems Support
     //                      First release
     //                      ENO used for internal error handling, interface has error and status
     //                      temp tag naming, insert constant
     // 03.00.00 23.04.2020  Simatic Systems Support
     //                      Set version to V3.0.0, harmonize the version of the whole library
     // 03.00.01 19.01.2020  Simatic Systems Support
     //                      Insert documentation
     //=============================================================================
   END_REGION BLOCK INFO HEADER

   REGION INITIALISATION
     #tempDate := #date;
     #tempDaysPassed := 0;
   END_REGION

   REGION COUNT DAYS
     // Check #date
     // adding zero forces the PLC to update the tag and eno check
     #tempDate := #tempDate + #TIME_ZERO_FORCE_UPDATE;
     IF ENO = FALSE THEN
       #error := TRUE;
       #status := #ERR_LIM_DATE;
       #LGF_GetCalendarDay := #tempDaysPassed;
       RETURN;
     END_IF;

     // Weekday of 1st January in the current year
     #tempDate.MONTH := #JANUARY;
     #tempDate.DAY := #FIRST_DAY;
     // adding zero forces the PLC to update the tag
     // in this case especially the weekday
     #tempDate := #tempDate + #TIME_ZERO_FORCE_UPDATE;

     // Days passed in the year since 1st January, "date" included
     #tempDaysPassed := DATE_TO_DINT(DTL_TO_DATE(#date)) - DATE_TO_DINT(DTL_TO_DATE(#tempDate)) + #ONE_DAY;
   END_REGION

   REGION OUTPUTS
     #error := FALSE;
     #status := #STATUS_NO_ERROR;
     #LGF_GetCalendarDay := #tempDaysPassed;

     // ENO is not used, forced to TRUE
     ENO := TRUE;
   END_REGION
END_FUNCTION